(* CODESYS project ShopFloorPLCLogic

Project tree, tasks and I/O mapping:
  Device : CODESYS Control Win V3 x64, CODESYS, version 3.5.20.40
    application Application
      libraries: Standard, 3.5.18.0 (System)
      task MainTask (cyclic, interval t#20ms, priority 1) calls PLC_PRG, SCADA_PRG
      function block Linear_Conveyor [SFC]
      function block Maq_3tools [ST]
      program PLC_PRG [CFC]
      program SCADA_PRG [ST]
      function block Warehouse [ST]
      function block Warehouse_In_Conveyor [ST]
      data type Warehouse_In_State
    Ethernet : Ethernet, CODESYS, version 4.2.0.0
      Modbus_TCP_Master : Modbus TCP Client, CODESYS, version 4.4.0.0
          settings: AutoReconnect = TRUE
        Modbus_TCP_Slave : Modbus TCP Slave, 3S - Smart Software Solutions GmbH, version 4.1.0.0
            settings: Unit-ID = 255; IPAddress = [192, 168, 1, 223]; Port = 5502; Channel 0.Function Code = 2; Channel 0.Read Offset = 16#0000; Channel 0.Read Length = 131; Channel 0.Write Offset = 0; Channel 0.Write Length = 0; Channel 0.Cycle Time = 100; Channel 1.Function Code = 15; Channel 1.Read Offset = 0; Channel 1.Read Length = 0; Channel 1.Write Offset = 16#0000; Channel 1.Write Length = 197; Channel 1.Cycle Time = 100; Channel 2.Function Code = 16; Channel 2.Read Offset = 0; Channel 2.Read Length = 0; Channel 2.Write Offset = 16#0000; Channel 2.Write Length = 1; Channel 2.Cycle Time = 100
            input  Cin1Sensor_0 : BOOL  // Channel 0.Channel 0.Bit0
            input  Cin2Sensor_0 : BOOL  // Channel 0.Channel 0.Bit1
            input  Cin3Sensor_0 : BOOL  // Channel 0.Channel 0.Bit2
            input  Cin4Sensor_0 : BOOL  // Channel 0.Channel 0.Bit3
            input  AT1_in0Sensor_0 : BOOL  // Channel 0.Channel 0.Bit4
            input  AT1_in1Sensor_0 : BOOL  // Channel 0.Channel 0.Bit5
            input  AT1_in2Sensor_0 : BOOL  // Channel 0.Channel 0.Bit6
            input  AT1_in3Sensor_0 : BOOL  // Channel 0.Channel 0.Bit7
            input  AT1_in4Sensor_0 : BOOL  // Channel 0.Channel 0.Bit0
            input  AT1_out1Sensor_0 : BOOL  // Channel 0.Channel 0.Bit1
            input  AT1_out2Sensor_0 : BOOL  // Channel 0.Channel 0.Bit2
            input  AT1_out3Sensor_0 : BOOL  // Channel 0.Channel 0.Bit3
            input  AT1_out4Sensor_0 : BOOL  // Channel 0.Channel 0.Bit4
            input  AT1_out5Sensor_0 : BOOL  // Channel 0.Channel 0.Bit5
            input  AT1_out6Sensor_0 : BOOL  // Channel 0.Channel 0.Bit6
            input  AT2_out0Sensor_0 : BOOL  // Channel 0.Channel 0.Bit7
            input  AT2_out1Sensor_0 : BOOL  // Channel 0.Channel 0.Bit0
            input  AT2_out2Sensor_0 : BOOL  // Channel 0.Channel 0.Bit1
            input  AT2_out3Sensor_0 : BOOL  // Channel 0.Channel 0.Bit2
            input  AT2_out4Sensor_0 : BOOL  // Channel 0.Channel 0.Bit3
            input  AT2_in1Sensor_0 : BOOL  // Channel 0.Channel 0.Bit4
            input  AT2_in2Sensor_0 : BOOL  // Channel 0.Channel 0.Bit5
            input  AT2_in3Sensor_0 : BOOL  // Channel 0.Channel 0.Bit6
            input  AT2_in4Sensor_0 : BOOL  // Channel 0.Channel 0.Bit7
            input  AT2_in5Sensor_0 : BOOL  // Channel 0.Channel 0.Bit0
            input  AT2_in6Sensor_0 : BOOL  // Channel 0.Channel 0.Bit1
            input  Cell0_CtopSensor_0 : BOOL  // Channel 0.Channel 0.Bit2
            input  Cell0_CmidSensor_0 : BOOL  // Channel 0.Channel 0.Bit3
            input  Cell0_CbotSensor_0 : BOOL  // Channel 0.Channel 0.Bit4
            input  Cell1_MtopSensor_0 : BOOL  // Channel 0.Channel 0.Bit5
            input  Cell1_MtopTool_Sensor : BOOL  // Channel 0.Channel 0.Bit6
            input  Cell1_MtopY_minus_Sensor : BOOL  // Channel 0.Channel 0.Bit7
            input  Cell1_MtopY_plus_Sensor : BOOL  // Channel 0.Channel 0.Bit0
            input  Cell1_MtopZ_minus_Sensor : BOOL  // Channel 0.Channel 0.Bit1
            input  Cell1_MtopZ_plus_Sensor : BOOL  // Channel 0.Channel 0.Bit2
            input  Cell1_CmidSensor_0 : BOOL  // Channel 0.Channel 0.Bit3
            input  Cell1_MbotSensor_0 : BOOL  // Channel 0.Channel 0.Bit4
            input  Cell1_MbotTool_Sensor : BOOL  // Channel 0.Channel 0.Bit5
            input  Cell1_MbotY_minus_Sensor : BOOL  // Channel 0.Channel 0.Bit6
            input  Cell1_MbotY_plus_Sensor : BOOL  // Channel 0.Channel 0.Bit7
            input  Cell1_MbotZ_minus_Sensor : BOOL  // Channel 0.Channel 0.Bit0
            input  Cell1_MbotZ_plus_Sensor : BOOL  // Channel 0.Channel 0.Bit1
            input  Cell2_MtopSensor_0 : BOOL  // Channel 0.Channel 0.Bit2
            input  Cell2_MtopTool_Sensor : BOOL  // Channel 0.Channel 0.Bit3
            input  Cell2_MtopY_minus_Sensor : BOOL  // Channel 0.Channel 0.Bit4
            input  Cell2_MtopY_plus_Sensor : BOOL  // Channel 0.Channel 0.Bit5
            input  Cell2_MtopZ_minus_Sensor : BOOL  // Channel 0.Channel 0.Bit6
            input  Cell2_MtopZ_plus_Sensor : BOOL  // Channel 0.Channel 0.Bit7
            input  Cell2_CmidSensor_0 : BOOL  // Channel 0.Channel 0.Bit0
            input  Cell2_MbotSensor_0 : BOOL  // Channel 0.Channel 0.Bit1
            input  Cell2_MbotTool_Sensor : BOOL  // Channel 0.Channel 0.Bit2
            input  Cell2_MbotY_minus_Sensor : BOOL  // Channel 0.Channel 0.Bit3
            input  Cell2_MbotY_plus_Sensor : BOOL  // Channel 0.Channel 0.Bit4
            input  Cell2_MbotZ_minus_Sensor : BOOL  // Channel 0.Channel 0.Bit5
            input  Cell2_MbotZ_plus_Sensor : BOOL  // Channel 0.Channel 0.Bit6
            input  Cell3_MtopSensor_0 : BOOL  // Channel 0.Channel 0.Bit7
            input  Cell3_MtopTool_Sensor : BOOL  // Channel 0.Channel 0.Bit0
            input  Cell3_MtopY_minus_Sensor : BOOL  // Channel 0.Channel 0.Bit1
            input  Cell3_MtopY_plus_Sensor : BOOL  // Channel 0.Channel 0.Bit2
            input  Cell3_MtopZ_minus_Sensor : BOOL  // Channel 0.Channel 0.Bit3
            input  Cell3_MtopZ_plus_Sensor : BOOL  // Channel 0.Channel 0.Bit4
            input  Cell3_CmidSensor_0 : BOOL  // Channel 0.Channel 0.Bit5
            input  Cell3_MbotSensor_0 : BOOL  // Channel 0.Channel 0.Bit6
            input  Cell3_MbotTool_Sensor : BOOL  // Channel 0.Channel 0.Bit7
            input  Cell3_MbotY_minus_Sensor : BOOL  // Channel 0.Channel 0.Bit0
            input  Cell3_MbotY_plus_Sensor : BOOL  // Channel 0.Channel 0.Bit1
            input  Cell3_MbotZ_minus_Sensor : BOOL  // Channel 0.Channel 0.Bit2
            input  Cell3_MbotZ_plus_Sensor : BOOL  // Channel 0.Channel 0.Bit3
            input  Cell4_MtopSensor_0 : BOOL  // Channel 0.Channel 0.Bit4
            input  Cell4_MtopTool_Sensor : BOOL  // Channel 0.Channel 0.Bit5
            input  Cell4_MtopY_minus_Sensor : BOOL  // Channel 0.Channel 0.Bit6
            input  Cell4_MtopY_plus_Sensor : BOOL  // Channel 0.Channel 0.Bit7
            input  Cell4_MtopZ_minus_Sensor : BOOL  // Channel 0.Channel 0.Bit0
            input  Cell4_MtopZ_plus_Sensor : BOOL  // Channel 0.Channel 0.Bit1
            input  Cell4_CmidSensor_0 : BOOL  // Channel 0.Channel 0.Bit2
            input  Cell4_MbotSensor_0 : BOOL  // Channel 0.Channel 0.Bit3
            input  Cell4_MbotTool_Sensor : BOOL  // Channel 0.Channel 0.Bit4
            input  Cell4_MbotY_minus_Sensor : BOOL  // Channel 0.Channel 0.Bit5
            input  Cell4_MbotY_plus_Sensor : BOOL  // Channel 0.Channel 0.Bit6
            input  Cell4_MbotZ_minus_Sensor : BOOL  // Channel 0.Channel 0.Bit7
            input  Cell4_MbotZ_plus_Sensor : BOOL  // Channel 0.Channel 0.Bit0
            input  Cell5_MtopSensor_0 : BOOL  // Channel 0.Channel 0.Bit1
            input  Cell5_MtopTool_Sensor : BOOL  // Channel 0.Channel 0.Bit2
            input  Cell5_MtopY_minus_Sensor : BOOL  // Channel 0.Channel 0.Bit3
            input  Cell5_MtopY_plus_Sensor : BOOL  // Channel 0.Channel 0.Bit4
            input  Cell5_MtopZ_minus_Sensor : BOOL  // Channel 0.Channel 0.Bit5
            input  Cell5_MtopZ_plus_Sensor : BOOL  // Channel 0.Channel 0.Bit6
            input  Cell5_CmidSensor_0 : BOOL  // Channel 0.Channel 0.Bit7
            input  Cell5_MbotSensor_0 : BOOL  // Channel 0.Channel 0.Bit0
            input  Cell5_MbotTool_Sensor : BOOL  // Channel 0.Channel 0.Bit1
            input  Cell5_MbotY_minus_Sensor : BOOL  // Channel 0.Channel 0.Bit2
            input  Cell5_MbotY_plus_Sensor : BOOL  // Channel 0.Channel 0.Bit3
            input  Cell5_MbotZ_minus_Sensor : BOOL  // Channel 0.Channel 0.Bit4
            input  Cell5_MbotZ_plus_Sensor : BOOL  // Channel 0.Channel 0.Bit5
            input  Cell6_MtopSensor_0 : BOOL  // Channel 0.Channel 0.Bit6
            input  Cell6_MtopTool_Sensor : BOOL  // Channel 0.Channel 0.Bit7
            input  Cell6_MtopY_minus_Sensor : BOOL  // Channel 0.Channel 0.Bit0
            input  Cell6_MtopY_plus_Sensor : BOOL  // Channel 0.Channel 0.Bit1
            input  Cell6_MtopZ_minus_Sensor : BOOL  // Channel 0.Channel 0.Bit2
            input  Cell6_MtopZ_plus_Sensor : BOOL  // Channel 0.Channel 0.Bit3
            input  Cell6_CmidSensor_0 : BOOL  // Channel 0.Channel 0.Bit4
            input  Cell6_MbotSensor_0 : BOOL  // Channel 0.Channel 0.Bit5
            input  Cell6_MbotTool_Sensor : BOOL  // Channel 0.Channel 0.Bit6
            input  Cell6_MbotY_minus_Sensor : BOOL  // Channel 0.Channel 0.Bit7
            input  Cell6_MbotY_plus_Sensor : BOOL  // Channel 0.Channel 0.Bit0
            input  Cell6_MbotZ_minus_Sensor : BOOL  // Channel 0.Channel 0.Bit1
            input  Cell6_MbotZ_plus_Sensor : BOOL  // Channel 0.Channel 0.Bit2
            input  Roll1aSensor_0 : BOOL  // Channel 0.Channel 0.Bit3
            input  Roll1bSensor_0 : BOOL  // Channel 0.Channel 0.Bit4
            input  Roll1cSensor_0 : BOOL  // Channel 0.Channel 0.Bit5
            input  Roll1dSensor_0 : BOOL  // Channel 0.Channel 0.Bit6
            input  Roll1eSensor_0 : BOOL  // Channel 0.Channel 0.Bit7
            input  Roll1fSensor_0 : BOOL  // Channel 0.Channel 0.Bit0
            input  Roll2aSensor_0 : BOOL  // Channel 0.Channel 0.Bit1
            input  Roll2bSensor_0 : BOOL  // Channel 0.Channel 0.Bit2
            input  Roll2cSensor_0 : BOOL  // Channel 0.Channel 0.Bit3
            input  Roll2dSensor_0 : BOOL  // Channel 0.Channel 0.Bit4
            input  Roll2eSensor_0 : BOOL  // Channel 0.Channel 0.Bit5
            input  Roll2fSensor_0 : BOOL  // Channel 0.Channel 0.Bit6
            input  Roll3aSensor_0 : BOOL  // Channel 0.Channel 0.Bit7
            input  Roll3bSensor_0 : BOOL  // Channel 0.Channel 0.Bit0
            input  Roll3cSensor_0 : BOOL  // Channel 0.Channel 0.Bit1
            input  Roll3dSensor_0 : BOOL  // Channel 0.Channel 0.Bit2
            input  Roll3eSensor_0 : BOOL  // Channel 0.Channel 0.Bit3
            input  Roll3fSensor_0 : BOOL  // Channel 0.Channel 0.Bit4
            input  Roll4aSensor_0 : BOOL  // Channel 0.Channel 0.Bit5
            input  Roll4bSensor_0 : BOOL  // Channel 0.Channel 0.Bit6
            input  Roll4cSensor_0 : BOOL  // Channel 0.Channel 0.Bit7
            input  Roll4dSensor_0 : BOOL  // Channel 0.Channel 0.Bit0
            input  Roll4eSensor_0 : BOOL  // Channel 0.Channel 0.Bit1
            input  Roll4fSensor_0 : BOOL  // Channel 0.Channel 0.Bit2
            output Cin1Motor_plus : BOOL  // Channel 1.Channel 1.Bit0
            output Cin1Motor_minus : BOOL  // Channel 1.Channel 1.Bit1
            output Cin2Motor_plus : BOOL  // Channel 1.Channel 1.Bit2
            output Cin2Motor_minus : BOOL  // Channel 1.Channel 1.Bit3
            output Cin3Motor_plus : BOOL  // Channel 1.Channel 1.Bit4
            output Cin3Motor_minus : BOOL  // Channel 1.Channel 1.Bit5
            output Cin4Motor_plus : BOOL  // Channel 1.Channel 1.Bit6
            output Cin4Motor_minus : BOOL  // Channel 1.Channel 1.Bit7
            output AT1_in0Motor_plus : BOOL  // Channel 1.Channel 1.Bit0
            output AT1_in0Motor_minus : BOOL  // Channel 1.Channel 1.Bit1
            output AT1_in0Warehouse_In : BOOL  // Channel 1.Channel 1.Bit2
            output AT1_in1Motor_plus : BOOL  // Channel 1.Channel 1.Bit3
            output AT1_in1Motor_minus : BOOL  // Channel 1.Channel 1.Bit4
            output AT1_in1Warehouse_In : BOOL  // Channel 1.Channel 1.Bit5
            output AT1_in2Motor_plus : BOOL  // Channel 1.Channel 1.Bit6
            output AT1_in2Motor_minus : BOOL  // Channel 1.Channel 1.Bit7
            output AT1_in2Warehouse_In : BOOL  // Channel 1.Channel 1.Bit0
            output AT1_in3Motor_plus : BOOL  // Channel 1.Channel 1.Bit1
            output AT1_in3Motor_minus : BOOL  // Channel 1.Channel 1.Bit2
            output AT1_in3Warehouse_In : BOOL  // Channel 1.Channel 1.Bit3
            output AT1_in4Motor_plus : BOOL  // Channel 1.Channel 1.Bit4
            output AT1_in4Motor_minus : BOOL  // Channel 1.Channel 1.Bit5
            output AT1_in4Warehouse_In : BOOL  // Channel 1.Channel 1.Bit6
            output AT1_out1Motor_plus : BOOL  // Channel 1.Channel 1.Bit7
            output AT1_out1Motor_minus : BOOL  // Channel 1.Channel 1.Bit0
            output AT1_out2Motor_plus : BOOL  // Channel 1.Channel 1.Bit1
            output AT1_out2Motor_minus : BOOL  // Channel 1.Channel 1.Bit2
            output AT1_out3Motor_plus : BOOL  // Channel 1.Channel 1.Bit3
            output AT1_out3Motor_minus : BOOL  // Channel 1.Channel 1.Bit4
            output AT1_out4Motor_plus : BOOL  // Channel 1.Channel 1.Bit5
            output AT1_out4Motor_minus : BOOL  // Channel 1.Channel 1.Bit6
            output AT1_out5Motor_plus : BOOL  // Channel 1.Channel 1.Bit7
            output AT1_out5Motor_minus : BOOL  // Channel 1.Channel 1.Bit0
            output AT1_out6Motor_plus : BOOL  // Channel 1.Channel 1.Bit1
            output AT1_out6Motor_minus : BOOL  // Channel 1.Channel 1.Bit2
            output AT2_out0Motor_plus : BOOL  // Channel 1.Channel 1.Bit3
            output AT2_out0Motor_minus : BOOL  // Channel 1.Channel 1.Bit4
            output AT2_out1Motor_plus : BOOL  // Channel 1.Channel 1.Bit5
            output AT2_out1Motor_minus : BOOL  // Channel 1.Channel 1.Bit6
            output AT2_out2Motor_plus : BOOL  // Channel 1.Channel 1.Bit7
            output AT2_out2Motor_minus : BOOL  // Channel 1.Channel 1.Bit0
            output AT2_out3Motor_plus : BOOL  // Channel 1.Channel 1.Bit1
            output AT2_out3Motor_minus : BOOL  // Channel 1.Channel 1.Bit2
            output AT2_out4Motor_plus : BOOL  // Channel 1.Channel 1.Bit3
            output AT2_out4Motor_minus : BOOL  // Channel 1.Channel 1.Bit4
            output AT2_in1Motor_plus : BOOL  // Channel 1.Channel 1.Bit5
            output AT2_in1Motor_minus : BOOL  // Channel 1.Channel 1.Bit6
            output AT2_in1Warehouse_In : BOOL  // Channel 1.Channel 1.Bit7
            output AT2_in2Motor_plus : BOOL  // Channel 1.Channel 1.Bit0
            output AT2_in2Motor_minus : BOOL  // Channel 1.Channel 1.Bit1
            output AT2_in2Warehouse_In : BOOL  // Channel 1.Channel 1.Bit2
            output AT2_in3Motor_plus : BOOL  // Channel 1.Channel 1.Bit3
            output AT2_in3Motor_minus : BOOL  // Channel 1.Channel 1.Bit4
            output AT2_in3Warehouse_In : BOOL  // Channel 1.Channel 1.Bit5
            output AT2_in4Motor_plus : BOOL  // Channel 1.Channel 1.Bit6
            output AT2_in4Motor_minus : BOOL  // Channel 1.Channel 1.Bit7
            output AT2_in4Warehouse_In : BOOL  // Channel 1.Channel 1.Bit0
            output AT2_in5Motor_plus : BOOL  // Channel 1.Channel 1.Bit1
            output AT2_in5Motor_minus : BOOL  // Channel 1.Channel 1.Bit2
            output AT2_in5Warehouse_In : BOOL  // Channel 1.Channel 1.Bit3
            output AT2_in6Motor_plus : BOOL  // Channel 1.Channel 1.Bit4
            output AT2_in6Motor_minus : BOOL  // Channel 1.Channel 1.Bit5
            output AT2_in6Warehouse_In : BOOL  // Channel 1.Channel 1.Bit6
            output Cell0_CtopMotor_plus : BOOL  // Channel 1.Channel 1.Bit7
            output Cell0_CtopMotor_minus : BOOL  // Channel 1.Channel 1.Bit0
            output Cell0_CmidMotor_plus : BOOL  // Channel 1.Channel 1.Bit1
            output Cell0_CmidMotor_minus : BOOL  // Channel 1.Channel 1.Bit2
            output Cell0_CbotMotor_plus : BOOL  // Channel 1.Channel 1.Bit3
            output Cell0_CbotMotor_minus : BOOL  // Channel 1.Channel 1.Bit4
            output Cell1_MtopMotor_plus : BOOL  // Channel 1.Channel 1.Bit5
            output Cell1_MtopMotor_minus : BOOL  // Channel 1.Channel 1.Bit6
            output Cell1_MtopRotate_minus : BOOL  // Channel 1.Channel 1.Bit7
            output Cell1_MtopRotate_plus : BOOL  // Channel 1.Channel 1.Bit0
            output Cell1_MtopTool : BOOL  // Channel 1.Channel 1.Bit1
            output Cell1_MtopY_minus : BOOL  // Channel 1.Channel 1.Bit2
            output Cell1_MtopY_plus : BOOL  // Channel 1.Channel 1.Bit3
            output Cell1_MtopZ_minus : BOOL  // Channel 1.Channel 1.Bit4
            output Cell1_MtopZ_plus : BOOL  // Channel 1.Channel 1.Bit5
            output Cell1_CmidMotor_plus : BOOL  // Channel 1.Channel 1.Bit6
            output Cell1_CmidMotor_minus : BOOL  // Channel 1.Channel 1.Bit7
            output Cell1_MbotMotor_plus : BOOL  // Channel 1.Channel 1.Bit0
            output Cell1_MbotMotor_minus : BOOL  // Channel 1.Channel 1.Bit1
            output Cell1_MbotRotate_minus : BOOL  // Channel 1.Channel 1.Bit2
            output Cell1_MbotRotate_plus : BOOL  // Channel 1.Channel 1.Bit3
            output Cell1_MbotTool : BOOL  // Channel 1.Channel 1.Bit4
            output Cell1_MbotY_minus : BOOL  // Channel 1.Channel 1.Bit5
            output Cell1_MbotY_plus : BOOL  // Channel 1.Channel 1.Bit6
            output Cell1_MbotZ_minus : BOOL  // Channel 1.Channel 1.Bit7
            output Cell1_MbotZ_plus : BOOL  // Channel 1.Channel 1.Bit0
            output Cell2_MtopMotor_plus : BOOL  // Channel 1.Channel 1.Bit1
            output Cell2_MtopMotor_minus : BOOL  // Channel 1.Channel 1.Bit2
            output Cell2_MtopRotate_minus : BOOL  // Channel 1.Channel 1.Bit3
            output Cell2_MtopRotate_plus : BOOL  // Channel 1.Channel 1.Bit4
            output Cell2_MtopTool : BOOL  // Channel 1.Channel 1.Bit5
            output Cell2_MtopY_minus : BOOL  // Channel 1.Channel 1.Bit6
            output Cell2_MtopY_plus : BOOL  // Channel 1.Channel 1.Bit7
            output Cell2_MtopZ_minus : BOOL  // Channel 1.Channel 1.Bit0
            output Cell2_MtopZ_plus : BOOL  // Channel 1.Channel 1.Bit1
            output Cell2_CmidMotor_plus : BOOL  // Channel 1.Channel 1.Bit2
            output Cell2_CmidMotor_minus : BOOL  // Channel 1.Channel 1.Bit3
            output Cell2_MbotMotor_plus : BOOL  // Channel 1.Channel 1.Bit4
            output Cell2_MbotMotor_minus : BOOL  // Channel 1.Channel 1.Bit5
            output Cell2_MbotRotate_minus : BOOL  // Channel 1.Channel 1.Bit6
            output Cell2_MbotRotate_plus : BOOL  // Channel 1.Channel 1.Bit7
            output Cell2_MbotTool : BOOL  // Channel 1.Channel 1.Bit0
            output Cell2_MbotY_minus : BOOL  // Channel 1.Channel 1.Bit1
            output Cell2_MbotY_plus : BOOL  // Channel 1.Channel 1.Bit2
            output Cell2_MbotZ_minus : BOOL  // Channel 1.Channel 1.Bit3
            output Cell2_MbotZ_plus : BOOL  // Channel 1.Channel 1.Bit4
            output Cell3_MtopMotor_plus : BOOL  // Channel 1.Channel 1.Bit5
            output Cell3_MtopMotor_minus : BOOL  // Channel 1.Channel 1.Bit6
            output Cell3_MtopRotate_minus : BOOL  // Channel 1.Channel 1.Bit7
            output Cell3_MtopRotate_plus : BOOL  // Channel 1.Channel 1.Bit0
            output Cell3_MtopTool : BOOL  // Channel 1.Channel 1.Bit1
            output Cell3_MtopY_minus : BOOL  // Channel 1.Channel 1.Bit2
            output Cell3_MtopY_plus : BOOL  // Channel 1.Channel 1.Bit3
            output Cell3_MtopZ_minus : BOOL  // Channel 1.Channel 1.Bit4
            output Cell3_MtopZ_plus : BOOL  // Channel 1.Channel 1.Bit5
            output Cell3_CmidMotor_plus : BOOL  // Channel 1.Channel 1.Bit6
            output Cell3_CmidMotor_minus : BOOL  // Channel 1.Channel 1.Bit7
            output Cell3_MbotMotor_plus : BOOL  // Channel 1.Channel 1.Bit0
            output Cell3_MbotMotor_minus : BOOL  // Channel 1.Channel 1.Bit1
            output Cell3_MbotRotate_minus : BOOL  // Channel 1.Channel 1.Bit2
            output Cell3_MbotRotate_plus : BOOL  // Channel 1.Channel 1.Bit3
            output Cell3_MbotTool : BOOL  // Channel 1.Channel 1.Bit4
            output Cell3_MbotY_minus : BOOL  // Channel 1.Channel 1.Bit5
            output Cell3_MbotY_plus : BOOL  // Channel 1.Channel 1.Bit6
            output Cell3_MbotZ_minus : BOOL  // Channel 1.Channel 1.Bit7
            output Cell3_MbotZ_plus : BOOL  // Channel 1.Channel 1.Bit0
            output Cell4_MtopMotor_plus : BOOL  // Channel 1.Channel 1.Bit1
            output Cell4_MtopMotor_minus : BOOL  // Channel 1.Channel 1.Bit2
            output Cell4_MtopRotate_minus : BOOL  // Channel 1.Channel 1.Bit3
            output Cell4_MtopRotate_plus : BOOL  // Channel 1.Channel 1.Bit4
            output Cell4_MtopTool : BOOL  // Channel 1.Channel 1.Bit5
            output Cell4_MtopY_minus : BOOL  // Channel 1.Channel 1.Bit6
            output Cell4_MtopY_plus : BOOL  // Channel 1.Channel 1.Bit7
            output Cell4_MtopZ_minus : BOOL  // Channel 1.Channel 1.Bit0
            output Cell4_MtopZ_plus : BOOL  // Channel 1.Channel 1.Bit1
            output Cell4_CmidMotor_plus : BOOL  // Channel 1.Channel 1.Bit2
            output Cell4_CmidMotor_minus : BOOL  // Channel 1.Channel 1.Bit3
            output Cell4_MbotMotor_plus : BOOL  // Channel 1.Channel 1.Bit4
            output Cell4_MbotMotor_minus : BOOL  // Channel 1.Channel 1.Bit5
            output Cell4_MbotRotate_minus : BOOL  // Channel 1.Channel 1.Bit6
            output Cell4_MbotRotate_plus : BOOL  // Channel 1.Channel 1.Bit7
            output Cell4_MbotTool : BOOL  // Channel 1.Channel 1.Bit0
            output Cell4_MbotY_minus : BOOL  // Channel 1.Channel 1.Bit1
            output Cell4_MbotY_plus : BOOL  // Channel 1.Channel 1.Bit2
            output Cell4_MbotZ_minus : BOOL  // Channel 1.Channel 1.Bit3
            output Cell4_MbotZ_plus : BOOL  // Channel 1.Channel 1.Bit4
            output Cell5_MtopMotor_plus : BOOL  // Channel 1.Channel 1.Bit5
            output Cell5_MtopMotor_minus : BOOL  // Channel 1.Channel 1.Bit6
            output Cell5_MtopRotate_minus : BOOL  // Channel 1.Channel 1.Bit7
            output Cell5_MtopRotate_plus : BOOL  // Channel 1.Channel 1.Bit0
            output Cell5_MtopTool : BOOL  // Channel 1.Channel 1.Bit1
            output Cell5_MtopY_minus : BOOL  // Channel 1.Channel 1.Bit2
            output Cell5_MtopY_plus : BOOL  // Channel 1.Channel 1.Bit3
            output Cell5_MtopZ_minus : BOOL  // Channel 1.Channel 1.Bit4
            output Cell5_MtopZ_plus : BOOL  // Channel 1.Channel 1.Bit5
            output Cell5_CmidMotor_plus : BOOL  // Channel 1.Channel 1.Bit6
            output Cell5_CmidMotor_minus : BOOL  // Channel 1.Channel 1.Bit7
            output Cell5_MbotMotor_plus : BOOL  // Channel 1.Channel 1.Bit0
            output Cell5_MbotMotor_minus : BOOL  // Channel 1.Channel 1.Bit1
            output Cell5_MbotRotate_minus : BOOL  // Channel 1.Channel 1.Bit2
            output Cell5_MbotRotate_plus : BOOL  // Channel 1.Channel 1.Bit3
            output Cell5_MbotTool : BOOL  // Channel 1.Channel 1.Bit4
            output Cell5_MbotY_minus : BOOL  // Channel 1.Channel 1.Bit5
            output Cell5_MbotY_plus : BOOL  // Channel 1.Channel 1.Bit6
            output Cell5_MbotZ_minus : BOOL  // Channel 1.Channel 1.Bit7
            output Cell5_MbotZ_plus : BOOL  // Channel 1.Channel 1.Bit0
            output Cell6_MtopMotor_plus : BOOL  // Channel 1.Channel 1.Bit1
            output Cell6_MtopMotor_minus : BOOL  // Channel 1.Channel 1.Bit2
            output Cell6_MtopRotate_minus : BOOL  // Channel 1.Channel 1.Bit3
            output Cell6_MtopRotate_plus : BOOL  // Channel 1.Channel 1.Bit4
            output Cell6_MtopTool : BOOL  // Channel 1.Channel 1.Bit5
            output Cell6_MtopY_minus : BOOL  // Channel 1.Channel 1.Bit6
            output Cell6_MtopY_plus : BOOL  // Channel 1.Channel 1.Bit7
            output Cell6_MtopZ_minus : BOOL  // Channel 1.Channel 1.Bit0
            output Cell6_MtopZ_plus : BOOL  // Channel 1.Channel 1.Bit1
            output Cell6_CmidMotor_plus : BOOL  // Channel 1.Channel 1.Bit2
            output Cell6_CmidMotor_minus : BOOL  // Channel 1.Channel 1.Bit3
            output Cell6_MbotMotor_plus : BOOL  // Channel 1.Channel 1.Bit4
            output Cell6_MbotMotor_minus : BOOL  // Channel 1.Channel 1.Bit5
            output Cell6_MbotRotate_minus : BOOL  // Channel 1.Channel 1.Bit6
            output Cell6_MbotRotate_plus : BOOL  // Channel 1.Channel 1.Bit7
            output Cell6_MbotTool : BOOL  // Channel 1.Channel 1.Bit0
            output Cell6_MbotY_minus : BOOL  // Channel 1.Channel 1.Bit1
            output Cell6_MbotY_plus : BOOL  // Channel 1.Channel 1.Bit2
            output Cell6_MbotZ_minus : BOOL  // Channel 1.Channel 1.Bit3
            output Cell6_MbotZ_plus : BOOL  // Channel 1.Channel 1.Bit4
            output Roll1fMotor_plus : BOOL  // Channel 1.Channel 1.Bit5
            output Roll1fMotor_minus : BOOL  // Channel 1.Channel 1.Bit6
            output Roll2fMotor_plus : BOOL  // Channel 1.Channel 1.Bit7
            output Roll2fMotor_minus : BOOL  // Channel 1.Channel 1.Bit0
            output Roll3fMotor_plus : BOOL  // Channel 1.Channel 1.Bit1
            output Roll3fMotor_minus : BOOL  // Channel 1.Channel 1.Bit2
            output Roll4fMotor_plus : BOOL  // Channel 1.Channel 1.Bit3
            output Roll4fMotor_minus : BOOL  // Channel 1.Channel 1.Bit4
            output Cin1Warehouse_Out : BOOL  // Channel 2.Channel 2.Bit0
            output Cin2Warehouse_Out : BOOL  // Channel 2.Channel 2.Bit1
            output Cin3Warehouse_Out : BOOL  // Channel 2.Channel 2.Bit2
            output Cin4Warehouse_Out : BOOL  // Channel 2.Channel 2.Bit3
            output AT1_out1Warehouse_Out : BOOL  // Channel 2.Channel 2.Bit4
            output AT1_out2Warehouse_Out : BOOL  // Channel 2.Channel 2.Bit5
            output AT1_out3Warehouse_Out : BOOL  // Channel 2.Channel 2.Bit6
            output AT1_out4Warehouse_Out : BOOL  // Channel 2.Channel 2.Bit7
            output AT1_out5Warehouse_Out : BOOL  // Channel 2.Channel 2.Bit8
            output AT1_out6Warehouse_Out : BOOL  // Channel 2.Channel 2.Bit9
            output AT2_out0Warehouse_Out : BOOL  // Channel 2.Channel 2.Bit10
            output AT2_out1Warehouse_Out : BOOL  // Channel 2.Channel 2.Bit11
            output AT2_out2Warehouse_Out : BOOL  // Channel 2.Channel 2.Bit12
            output AT2_out3Warehouse_Out : BOOL  // Channel 2.Channel 2.Bit13
            output AT2_out4Warehouse_Out : BOOL  // Channel 2.Channel 2.Bit14
            unmapped channels: Channel 0, Channel 1, Channel 2
      ModbusTCP_Slave_Device : ModbusTCP Server Device, CODESYS, version 4.4.0.0
          settings: UpdateableHolding = TRUE; DistinctBitAreas = TRUE; Coils Size = 8; Discrete Inputs Size = 8
          output S_sensor1 : BOOL  // Holding Registers.Holding Registers.Bit0
          output S_sensor2 : BOOL  // Holding Registers.Holding Registers.Bit1
          output S_sensor3 : BOOL  // Holding Registers.Holding Registers.Bit2
          output C1_stop : BOOL  // Holding Registers.Holding Registers.Bit0
          output C2_stop : BOOL  // Holding Registers.Holding Registers.Bit1
          output C3_stop : BOOL  // Holding Registers.Holding Registers.Bit2
          output Gate0 : BOOL  // Coils.Coils.Bit0
          output Gate1 : BOOL  // Coils.Coils.Bit1
          output Gate2 : BOOL  // Coils.Coils.Bit2
          unmapped channels: Holding Registers, Input Registers, Coils, Discrete Inputs
*)

// Device/Application/Warehouse_In_State
{attribute 'qualified_only'}
{attribute 'strict'}
TYPE Warehouse_In_State :
(
	IDLE,
	WAIT_FOR_SHIT,
	TAKE_SHIT,
	SEND_SHIT
) INT := WAIT_FOR_SHIT;
END_TYPE

// Device/Application/PLC_PRG
PROGRAM PLC_PRG
VAR
	C1, C2, C3: Linear_Conveyor;
END_VAR

C1(sensor := Cell0_CtopSensor_0, free_I := C2.free_O, recv_I := Cell0_CtopSensor_0); // Linear_Conveyor
Cell0_CtopMotor_plus := C1.right;
C2(sensor := Cell0_CmidSensor_0, free_I := C3.free_O, recv_I := C1.recv_O); // Linear_Conveyor
Cell0_CmidMotor_plus := C2.right;
C3(sensor := Cell0_CbotSensor_0, free_I := false, recv_I := C2.recv_O); // Linear_Conveyor
Cell0_CbotMotor_plus := C3.right;

END_PROGRAM

// Device/Application/Linear_Conveyor
FUNCTION_BLOCK Linear_Conveyor
VAR_INPUT
	sensor: BOOL;
	free_I: BOOL;
	recv_I: BOOL;
END_VAR
VAR_OUTPUT
	right : BOOL;
	free_O: BOOL;
	recv_O: BOOL;
END_VAR
VAR
END_VAR

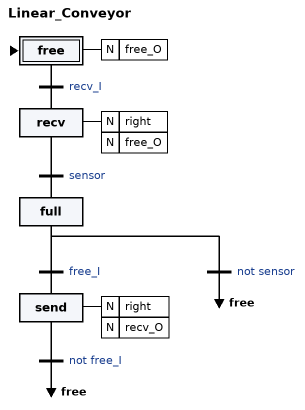
INITIAL_STEP free:
    free_O(N);
END_STEP
TRANSITION FROM free TO recv
    := recv_I;
END_TRANSITION
STEP recv:
    right(N);
    free_O(N);
END_STEP
TRANSITION FROM recv TO full
    := sensor;
END_TRANSITION
STEP full:
END_STEP
TRANSITION FROM full TO send
    := free_I;
END_TRANSITION
TRANSITION FROM full TO free
    := not sensor;
END_TRANSITION
STEP send:
    right(N);
    recv_O(N);
END_STEP
TRANSITION FROM send TO free
    := not free_I;
END_TRANSITION

END_FUNCTION_BLOCK

// Device/Application/SCADA_PRG
PROGRAM SCADA_PRG
VAR
END_VAR

Gate0 := Cell0_CtopMotor_plus;
Gate1 := Cell0_CmidMotor_plus;
Gate2 := Cell0_CbotMotor_plus;
S_sensor1 := Cell0_CtopSensor_0;
S_sensor2 := Cell0_CmidSensor_0;
S_sensor3 := Cell0_CbotSensor_0;
Cell0_CtopMotor_plus := Cell0_CtopMotor_plus AND (NOT C1_stop);
Cell0_CmidMotor_plus := Cell0_CmidMotor_plus AND (NOT C2_stop);
Cell0_CbotMotor_plus := Cell0_CbotMotor_plus AND (NOT C3_stop);

END_PROGRAM

// Device/Application/Maq_3tools
FUNCTION_BLOCK Maq_3tools
VAR_INPUT
END_VAR
VAR_OUTPUT
END_VAR
VAR
END_VAR

END_FUNCTION_BLOCK

// Device/Application/Warehouse
FUNCTION_BLOCK PUBLIC Warehouse
VAR_INPUT
    sensor1, sensor2, sensor3, sensor4 : BOOL;
END_VAR
VAR_OUTPUT
	motor1_plus, motor2_plus, motor3_plus, motor4_plus : BOOL;
END_VAR
VAR
	product_counter : INT;
END_VAR

IF sensor1 THEN
	motor1_plus := TRUE;
END_IF

END_FUNCTION_BLOCK

// Device/Application/Warehouse_In_Conveyor
FUNCTION_BLOCK Warehouse_In_Conveyor
VAR_INPUT
	sensor: BOOL;
	full_I: BOOL;
	recv_I: BOOL;
END_VAR
VAR_OUTPUT
	warehouse_in_O: BOOL;
	motor_plus: BOOL;
	free_O: BOOL;
END_VAR
VAR
	state: Warehouse_In_State;
END_VAR

CASE state OF
	Warehouse_In_State.WAIT_FOR_SHIT:
		free_O := TRUE;
		warehouse_in_O := FALSE;
		IF recv_I = 1 THEN
			state := Warehouse_In_State.TAKE_SHIT;
		END_IF
		IF sensor = 1 THEN
			state := Warehouse_In_State.SEND_SHIT;
		END_IF
	Warehouse_In_State.TAKE_SHIT:
		motor_plus := TRUE;
		IF sensor = 1 THEN
			state := Warehouse_In_State.SEND_SHIT;
		END_IF
	Warehouse_In_State.SEND_SHIT:
		motor_plus := FALSE;
		free_O := FALSE;
		IF  full_I = 0 THEN
			warehouse_in_O := TRUE;
			state := Warehouse_In_State.WAIT_FOR_SHIT;
		END_IF
END_CASE

END_FUNCTION_BLOCK
